// TIA Portal V20 export
TYPE "LConSMC_typeFrictionMeasurementV2In"
// stored: Access Published
   STRUCT
      execute : Bool;   // TRUE: Starte Messung mit steigender Flanke / TRUE: Start friction measurement with rising edge
      abort : Bool;   // TRUE: Stoppe Messung und Achse mit steigender Flanke / TRUE: Rising edge stops measurement and axis
      warmUpTime : Time;   // Warmlaufzeit Vor Beginn der Messung dreht der Antrieb für die parametrierte Zeit mit der maximalen Messdrehzahl / Warm up time Before the measurement starts the drive rotates with maximum measurement speed for the parameterized time
      rampTime : Real := 1000.0;   // [ms] Time to ramp up to maximum speed
      noOfMeasurementPoints : Int := 50;   // Anzahl an Messpunkten pro Drehzahlwert (Einstellbar zwischen 50-500) / Number measurement points per speed step (limited between 50-500)
      sizeOfArray : Int := 20;   // maxSpeed = 0: Anzahl der verwendeten Stützpunkte (aus "speedValues") maxSpeed <> 0: Anzahl an Messpunkten zwischen 0 und "maxSpeed" / maxSpeed = 0: Number of breakpoints (from "speedValues") maxSpeed <> 0: Number of measuring points between 0 and "maxSpeed"
      maxSpeed : LReal := 0.0;   // [1/min] Maximaldrehzahl für die die Reibung gemessen werden soll / [RPM] Maximim speed at which the friction should be recorded
      speedValues : "LConSMC_typeBreakPointTable";   // [1/min] Stützpunkte der Drehzahlwerte für die die Reibung gemessen werden soll. Wird nur verwendet wenn "maxSpeed" = 0. / [RPM] Breakpoints of speed values for which the friction should be measured. Only if "maxSpeed" = 0.
      measurementDelayTime : Time := T#1S;   // Einschwingzeit für jeden Messpunkt nachdem die Reibung gemessen wird / Settling time after which the friction is measured at each speed setpoint
   END_STRUCT;
   // speedValues.values[0..19] := 0.0;
END_TYPE
